{attribute 'GeneratedUsingTerminal: EL6751--0000'}
{attribute addProperty BoxType "EL6751--0000"}
{attribute addProperty Description "EL6751 CANopen Master (HW-Version 01)"}
{attribute addProperty Physics "KK"}
{attribute addProperty Id "InfoDataAT %I*InfoData_90184F0C16"}
{attribute addProperty CRC "554310285"}
{attribute addProperty Size "16"}
TYPE EL6751_210A1A8D EXTENDS EtcSlaveTerminalBase_947E5A46 :
STRUCT
	{attribute addProperty Name "InfoData"}
	InfoData : InfoData_90184F0C;
END_STRUCT
END_TYPE

(* stored: Version 1.2.0.0, ProductVersion 3.1.4024.11
   DUT EL6751_210A1A8D: Id {f68a659a-0c57-49e9-9a9b-b085c1bd0ddb} *)
